// TwinCAT 3 PLC project Caller
// ProgramVersion: 3.1.4023.0
// libraries:
//   Tc2_DataExchange, * (Beckhoff Automation GmbH)
//   Tc2_Standard, * (Beckhoff Automation GmbH)
//   Tc2_System, * (Beckhoff Automation GmbH)
//   Tc2_Utilities, * (Beckhoff Automation GmbH)
//   Tc3_Module, * (Beckhoff Automation GmbH)
// project tree:
//   Code/ F_GetAmsNetId.TcPOU (not stored), I_Executable.TcIO (not stored), I_Logger.TcIO (not stored), ST_AdsReadWriteOptions.TcDUT (not stored), ST_SymbolHandle.TcDUT (not stored), ST_SymbolAddress.TcDUT (not stored), T_AdsWrite.TcPOU, T_GetLastMsgLogger.TcPOU, T_ReleaseHandle.TcPOU, T_GetHandle.TcPOU, T_CallMethod.TcPOU, T_AdsReadWrite.TcPOU, T_InvokeRpcMethod.TcPOU
//   / PlcTask.TcTTO
//   POUs/ FB_InvokeRpcMethod.TcPOU, MAIN.TcPOU
// (motion and I/O tree: see PLC project provider)
// real-time tasks:
//   TASK PlcTask: cycle T#10ms, priority 20, ADS port 350
//   TASK PlcTask1: cycle T#10ms, priority 21, ADS port 351

CONFIGURATION Caller
    RESOURCE PLC ON TwinCAT3
        TASK PlcTask(INTERVAL := T#10ms, PRIORITY := 21);
        PROGRAM MAIN WITH PlcTask : MAIN;
    END_RESOURCE
END_CONFIGURATION

// ---- POUs/MAIN.TcPOU
PROGRAM MAIN
VAR
   xCall : BOOL;
   AddParams : M_ADD_Parameters := (A := 40, B := 2);
   MeaningOfLife : LREAL;
	
	
	askForTheOdds : BOOL;
   c3poAddition : M_ADD_Parameters := (A := 3000, B := 720);
   OddsOfNavigatingAnAsteroidField : LREAL;
	C3PO_Says : STRING(255);

   fbRPC : FB_InvokeRpcMethod;
   invokeRpc : T_InvokeRpcMethod;
   xBusy : BOOL;
   xError : BOOL;
   nErrorID : UDINT;
   methodHandle : ST_SymbolHandle;
   taskState : I_Executable;
   invokeDone, invokeError, invokeBusy : BOOL;
	doneRt, errRt, busyRt : R_TRIG;
   logger : T_GetLastMsgLogger;
   firstScan : BOOL := TRUE;
	
	
END_VAR
VAR CONSTANT
	EMPTY_STRING : STRING := '';
	C3PO_ERR_MSG : STRING(255) := 'Sir, I don$'t know where your ship learned to communicate, but it has the most peculiar dialect.';
END_VAR

fbRPC(
	bCall:=xCall , 
	sNetId :='' , 
	nPort :=851 , 
	sMethodName :='MAIN.fbMath#M_ADD' , 
	nSrcAddrParameter :=ADR(AddParams) , 
	nLenParameter :=SIZEOF(AddParams) , 
	nDestAddrReturnValue :=ADR(MeaningOfLife) , 
	nLenReturnValue :=SIZEOF(MeaningOfLife) , 
	tTimeout :=DEFAULT_ADS_TIMEOUT , 
	eComMode :=E_AdsComMode.eAdsComModeFastCom , 
	bBusy =>xBusy , 
	bError =>xError , 
	nErrorId =>nErrorID );

IF firstScan THEN
	firstScan := FALSE;
	invokeRpc.SetLogger(logger);
	
END_IF

logger.lastLog;
logger.lasLogLevel;
C3PO_Says;

invokeRpc();
methodHandle.SymbolAddress.Ads.netId := F_ScanAmsNetIds('0.0.0.0.0.0.0');
methodHandle.SymbolAddress.Ads.port := 851;
methodHandle.SymbolAddress.SymbolName := 'MAIN.fbMath#M_ADD';
methodHandle.SymbolAddress.WriteRef := F_BIGTYPE(pData := ADR(c3poAddition), cbLen := SIZEOF(c3poAddition));
methodHandle.SymbolAddress.ReadRef := F_LREAL(OddsOfNavigatingAnAsteroidField);

IF askForTheOdds THEN
   askForTheOdds := FALSE;
   taskState := 0;

   invokeRpc.TryInvokeMethodCall(
      symbolHandle := methodHandle,
      adsTimeout := DEFAULT_ADS_TIMEOUT,
      status => taskState
   );

END_IF

invokeBusy := taskState <> 0 AND_THEN taskState.Busy;
invokeDone := taskState <> 0 AND_THEN taskState.Done;
invokeError := taskState <> 0 AND_THEN taskState.Error;
busyRt( CLK := invokeBusy );
doneRt( CLK := invokeDone );
errRt( CLK := invokeError);

IF busyRt.Q THEN
	C3PO_Says := EMPTY_STRING;
END_IF

IF doneRt.Q  THEN
	C3PO_Says := CONCAT(
							'Sir, the possibility of successfully navigating an asteroid field is approximately ', 
							CONCAT( TO_STRING(TO_INT(OddsOfNavigatingAnAsteroidField)), ' to 1.')
						);
END_IF

IF errRt.Q  THEN
	C3PO_Says := C3PO_ERR_MSG;
END_IF

END_PROGRAM

// ---- POUs/FB_InvokeRpcMethod.TcPOU
{attribute 'hide_all_locals'}
FUNCTION_BLOCK FB_InvokeRpcMethod
VAR_INPUT
	bCall					: BOOL;
	sNetId					: T_AmsNetId;
	nPort					: T_AmsPort := 851;
	sMethodName				: STRING(255); //Example:MAIN.fbMath#M_ADD
	nSrcAddrParameter		: PVOID;
	nLenParameter			: UDINT;
	                          
	nDestAddrReturnValue	: PVOID;
	nLenReturnValue			: UDINT;
	                          
	tTimeout				: TIME := DEFAULT_ADS_TIMEOUT;
	eComMode				: E_AdsComMode := eAdsComModeSecureCom;
END_VAR                       
VAR_OUTPUT                    
	bBusy					: BOOL;
	bError					: BOOL;
	nErrorId				: UDINT;
END_VAR                       
VAR                           
	_sNetId					: T_AmsNetId;
 	_sMethodName			: STRING(255);	
	_nPort					: T_AmsPort;
	fbGetHandle				: ADSRDWRT;
	fbCallMethod			: ADSRDWRT;
	fbReleaseHandle			: ADSWRITE;
	trigCall				: R_TRIG;
	eStep,eNextStep			: (IDLE,GET_HANDLE,CALL_METHOD,RELEASE_HANDLE) :=IDLE ;
	nMethodHandle 			: DWORD := 0;
END_VAR

trigCall(CLK:=bCall);
CASE eStep OF
	IDLE:
		IF trigCall.Q THEN
			bBusy 				:= TRUE;
			nErrorId 			:= 0;
			bError 				:= FALSE;
			fbGetHandle			(WRTRD := FALSE);
			fbCallMethod		(WRTRD := FALSE);
			fbReleaseHandle		(WRITE := FALSE);
			IF nMethodHandle <> 0 THEN
				IF 	_sMethodName =  sMethodName AND
					_sNetId 	 = 	sNetId 		AND
					_nPort 		 = 	nPort
				THEN
					eStep			:= CALL_METHOD;
				ELSE        	
					eStep			:= RELEASE_HANDLE;
					eNextStep		:= GET_HANDLE;
				END_IF
			ELSE
				eStep	:=GET_HANDLE;
			END_IF
		ELSE
			bBusy := FALSE;
		END_IF
		
	GET_HANDLE:
		fbGetHandle(NETID 		:= sNetId,
					PORT 		:= nPort,
					IDXGRP 		:= ADSIGRP_SYM_HNDBYNAME,
					IDXOFFS 	:= 0,
					SRCADDR 	:= ADR(sMethodName),
					WRITELEN 	:= TO_UDINT(LEN(sMethodName)),
					DESTADDR 	:= ADR(nMethodHandle),
					READLEN 	:= SIZEOF(nMethodHandle),
					WRTRD 		:= TRUE,
					TMOUT 		:= tTimeout,
					ERR 		=> bError,
					ERRID 		=> nErrorId);

		IF NOT fbGetHandle.BUSY THEN
			IF NOT bError THEN
				_sMethodName 	:= sMethodName;
				_sNetId 		:= sNetId;
				_nPort 			:= nPort;
				eStep			:= CALL_METHOD;
			ELSE
				eStep			:= IDLE;
			END_IF
			fbGetHandle(WRTRD := FALSE);
		END_IF
		
	CALL_METHOD:
		fbCallMethod( NETID		:= sNetId , 
					  PORT		:= nPort , 
					  IDXGRP	:= ADSIGRP_SYM_VALBYHND , 
					  IDXOFFS	:= nMethodHandle , 
					  WRITELEN	:= nLenParameter , 
					  READLEN	:= nLenReturnValue , 
					  SRCADDR	:= nSrcAddrParameter , 
					  DESTADDR	:= nDestAddrReturnValue , 
					  WRTRD		:= TRUE , 
					  TMOUT		:= tTimeout , 
					  ERR		=> bError , 
					  ERRID		=> nErrorId );

		IF NOT fbCallMethod.Busy THEN
			IF NOT bError THEN
				IF (eComMode = eAdsComModeSecureCom) THEN
					eStep		:= RELEASE_HANDLE;
					eNextStep	:= IDLE;
				ELSE
					eStep		:= IDLE;
				END_IF
			ELSE
				eStep			:= RELEASE_HANDLE;
				eNextStep		:= IDLE;				
			END_IF
			fbCallMethod(WRTRD := FALSE);
		END_IF							 
							 
							 
	RELEASE_HANDLE:
		fbReleaseHandle(NETID 		:= sNetId,
						PORT 		:= nPort,
						IDXGRP 		:= ADSIGRP_SYM_RELEASEHND,
						IDXOFFS 	:= 0,
            SRCADDR := ADR(nMethodHandle),
            LEN := SIZEOF(nMethodHandle),
						LEN 		:= 0,
						WRITE 		:= TRUE,
						TMOUT 		:= tTimeout,
						ERR 		=> bError,
						ERRID 		=> nErrorId);

		IF NOT fbReleaseHandle.Busy THEN
			nMethodHandle 	:= 0;
			fbReleaseHandle	(Write := FALSE);
			eStep 			:= eNextStep;
		END_IF
	
END_CASE

END_FUNCTION_BLOCK

// ---- Code/T_InvokeRpcMethod.TcPOU
FUNCTION_BLOCK T_InvokeRpcMethod
VAR_INPUT
   bCall : BOOL;
   sNetId : T_AmsNetId;
   nPort : T_AmsPort := 851;
   sMethodName : STRING(255); //Example:MAIN.fbMath#M_ADD
   nSrcAddrParameter : PVOID;
   nLenParameter : UDINT;

   nDestAddrReturnValue : PVOID;
   nLenReturnValue : UDINT;

   tTimeout : TIME := DEFAULT_ADS_TIMEOUT;
   eComMode : E_AdsComMode := eAdsComModeSecureCom;
END_VAR
VAR_OUTPUT
   bBusy : BOOL;
   bError : BOOL;
   nErrorId : UDINT;
END_VAR
VAR
   getHandle : T_GetHandle;
   callMethod : T_CallMethod;
   releaseHandle : T_ReleaseHandle;
   symbolHandle : ST_SymbolHandle;

   _sNetId : T_AmsNetId;
   _sMethodName : STRING(255);
   _nPort : T_AmsPort;
   //	fbGetHandle				: ADSRDWRT;
   //	fbCallMethod			: ADSRDWRT;
   //	fbReleaseHandle			: ADSWRITE;
   trigCall : R_TRIG;
   eStep, prevStep : (
      IDLE,
      GET_HANDLE,
      CALL_METHOD,
      RELEASE_HANDLE
   ) := IDLE;
  status : I_Executable;
END_VAR

trigCall(CLK := bCall);

CASE eStep OF
   IDLE:
	
		prevStep := eStep;
      IF trigCall.Q THEN
         bBusy := TRUE;
         nErrorId := 0;
         bError := FALSE;
			
			symbolHandle.SymbolAddress.SymbolName := sMethodName;
			symbolHandle.Handle := 0;
			symbolHandle.SymbolAddress.Ads.netId := F_ScanAmsNetIds(sNetId);
			symbolHandle.SymbolAddress.Ads.port := nPort;
			
			symbolHandle.SymbolAddress.WriteRef.cbLen := nLenParameter;
			symbolHandle.SymbolAddress.WriteRef.pData := nSrcAddrParameter;
			
			symbolHandle.SymbolAddress.ReadRef.cbLen := nLenReturnValue;
			symbolHandle.SymbolAddress.ReadRef.pData := nDestAddrReturnValue;
			eStep := GET_HANDLE;
         
      ELSE
         bBusy := FALSE;
      END_IF

   GET_HANDLE:
      IF prevStep <> eStep THEN
			getHandle.TryGetHandle(symbolHandle, DEFAULT_ADS_TIMEOUT);
			prevStep := eStep;
			
		ELSE
			IF getHandle.Done THEN
				eStep := CALL_METHOD;
			END_IF
			
		END_IF

   CALL_METHOD:
	
      IF prevStep <> eStep THEN
			callMethod.TryMethodCall(symbolHandle, DEFAULT_ADS_TIMEOUT);
			prevStep := eStep;
			
		ELSE
			IF callMethod.Done THEN
				eStep := RELEASE_HANDLE;
			END_IF
			
		END_IF
      

   RELEASE_HANDLE:
      
		IF prevStep <> eStep THEN
			releaseHandle.TryReleaseHandle(symbolHandle, DEFAULT_ADS_TIMEOUT);
			prevStep := eStep;
			
		ELSE
			IF releaseHandle.Done THEN
				eStep := IDLE;
			END_IF
			
		END_IF

END_CASE

getHandle();
callMethod();
releaseHandle();

END_FUNCTION_BLOCK

// ---- Code/T_GetHandle.TcPOU
FUNCTION_BLOCK T_GetHandle IMPLEMENTS I_Executable
VAR
   logger : I_Logger;
   _symbolHandle : REFERENCE TO ST_SymbolHandle; // just for debug
	readWrite : T_AdsReadWrite;

END_VAR
VAR CONSTANT
   NO_ERR : UDINT := 0;
   LOG_DEBUG : DWORD := 0;
   LOG_INFO : DWORD := ADSLOG_MSGTYPE_HINT;
   LOG_WARNING : DWORD := ADSLOG_MSGTYPE_WARN;
   LOG_ERROR : DWORD := ADSLOG_MSGTYPE_ERROR;
END_VAR

readWrite();

PROPERTY Busy : BOOL
GET
Busy := readWrite.Busy;
END_GET
END_PROPERTY

PROPERTY Done : BOOL
GET
Done := readWrite.Done;
END_GET
END_PROPERTY

PROPERTY Error : BOOL
GET
Error := readWrite.Error;
END_GET
END_PROPERTY

METHOD PRIVATE ToLog
VAR_INPUT
	Msg : STRING(255);
	LogLevel : DWORD; // generic level, can be mapped to logging framework
END_VAR
IF logger = 0 THEN
	RETURN;
	
END_IF

logger.ToLog(Msg, LogLevel);
END_METHOD

METHOD TryGetHandle : BOOL
VAR_IN_OUT
	symbolHandle : ST_SymbolHandle; // This handle object will be used in the next step.
END_VAR
VAR_INPUT
	adsTimeout : TIME := DEFAULT_ADS_TIMEOUT; // DEFAULT_ADS_TIMEOUT is T#5s;
END_VAR
VAR_OUTPUT
	status : I_Executable;
END_VAR
VAR
	readWriteOpts : ST_AdsReadWriteOptions;
END_VAR
VAR CONSTANT
	NO_HANDLE : DWORD := 0;
END_VAR
IF Busy THEN
	ToLog('Cannot TryGetHandle as Busy', LOG_WARNING);
	RETURN;
	
END_IF

_symbolHandle REF= symbolHandle;

readWriteOpts.AdsAddress := symbolHandle.SymbolAddress.Ads;
readWriteOpts.IndexGroup := ADSIGRP_SYM_HNDBYNAME;
readWriteOpts.IndexOffset := 0;
readWriteOpts.WriteParams := F_STRING(symbolHandle.SymbolAddress.SymbolName);
readWriteOpts.ReadParams := F_DWORD(symbolHandle.Handle);
readWriteOpts.Timeout := adsTimeout;

TryGetHandle := readWrite.TryRequest( readWriteOpts, status => status );
END_METHOD

END_FUNCTION_BLOCK

// ---- Code/T_AdsReadWrite.TcPOU
FUNCTION_BLOCK T_AdsReadWrite IMPLEMENTS I_Executable
VAR
   logger : I_Logger;
	_readWriteOpts : ST_AdsReadWriteOptions;
	
   readWrite : ADSRDWRT;

   state, prevState : (
      IDLE,
      REQUEST,
      WAIT_FOR_RESPONSE,
      DONE_STATE,
      ERROR_STATE
   );

   lastErrorId : UDINT;

END_VAR
VAR CONSTANT
   NO_ERR : UDINT := 0;
   LOG_DEBUG : DWORD := 0;
   LOG_INFO : DWORD := ADSLOG_MSGTYPE_HINT;
   LOG_WARNING : DWORD := ADSLOG_MSGTYPE_WARN;
   LOG_ERROR : DWORD := ADSLOG_MSGTYPE_ERROR;
END_VAR

CASE state OF

   IDlE:
      IsEntryActionAndLog();

   REQUEST:
      IsEntryActionAndLog();
		
      lastErrorId := NO_ERR;
      readWrite.WRTRD := TRUE;
      state := WAIT_FOR_RESPONSE;

   WAIT_FOR_RESPONSE:
      IsEntryActionAndLog();

      IF readWrite.ERR THEN
         state := ERROR_STATE;

      ELSIF NOT readWrite.BUSY THEN
         state := DONE_STATE;

      END_IF

   DONE_STATE:
      IsEntryActionAndLog();

   ERROR_STATE:
      IF IsEntryActionAndLog() THEN
         lastErrorId := readWrite.ERRID;
			
      END_IF

END_CASE

readWrite.WRTRD R= NOT Busy;
readWrite();

PROPERTY Busy : BOOL
GET
Busy := 
	NOT Done 
	AND NOT Error 
	AND state <> IDLE;
END_GET
END_PROPERTY

PROPERTY Done : BOOL
GET
Done := state = DONE_STATE;
END_GET
END_PROPERTY

PROPERTY Error : BOOL
GET
Error := state = ERROR_STATE;
END_GET
END_PROPERTY

METHOD PRIVATE IsEntryActionAndLog : BOOL
IsEntryActionAndLog := prevState <> state;

// useful to debug state transitions. to avoid "chatter" LogFramework should have runtime log level switches 
// i.e. https://github.com/Intecre/twincat-utils/tree/master/IntecreUtilities/IntecreUtilities/IntecreUtilities/Utilities/Logger
// see also https://github.com/Intecre/twincat-utils/blob/master/IntecreUtilities/IntecreUtilities/IntecreUtilities/Utilities/T_NamedBase.TcPOU
ToLog(
	Msg := CONCAT(CONCAT(TO_STRING(prevState), ' transition to state '), TO_STRING(state)), 
	LogLevel:= LOG_DEBUG
);

prevState := state;
END_METHOD

METHOD PUBLIC SetLogger
VAR_INPUT
	logger : I_Logger;
END_VAR
THIS^.logger := logger;
END_METHOD

METHOD PRIVATE ToLog
VAR_INPUT
	Msg : STRING(255);
	LogLevel : DWORD; // generic level, can be mapped to logging framework
END_VAR
IF logger = 0 THEN
	RETURN;
	
END_IF

logger.ToLog(Msg, LogLevel);
END_METHOD

METHOD TryRequest : BOOL
VAR_INPUT
	readWriteOptions : ST_AdsReadWriteOptions;
END_VAR
VAR_OUTPUT
	status : I_Executable;
END_VAR
VAR CONSTANT
	NO_HANDLE : DWORD := 0;
END_VAR
IF Busy THEN
	ToLog('Cannot TryRequest as Busy', LOG_WARNING);
	RETURN;
	
END_IF

_readWriteOpts := readWriteOptions;
readWrite(
	NETID := F_GetAmsNetId(_readWriteOpts.AdsAddress.netId),
	PORT := _readWriteOpts.AdsAddress.port,
	IDXGRP := _readWriteOpts.IndexGroup,
	IDXOFFS := _readWriteOpts.IndexOffset,
	WRITELEN := _readWriteOpts.WriteParams.cbLen,
	SRCADDR := _readWriteOpts.WriteParams.pData,
	READLEN := _readWriteOpts.ReadParams.cbLen,
	DESTADDR := _readWriteOpts.ReadParams.pData,
	TMOUT := _readWriteOpts.Timeout
);

state := REQUEST;

TryRequest := TRUE;
status := THIS^;
END_METHOD

END_FUNCTION_BLOCK

// ---- Code/T_CallMethod.TcPOU
FUNCTION_BLOCK T_CallMethod IMPLEMENTS I_Executable
VAR
   logger : I_Logger;
	_symbolHandle : ST_SymbolHandle;
	readWrite : T_AdsReadWrite;
END_VAR
VAR CONSTANT
   LOG_DEBUG : DWORD := 0;
   LOG_INFO : DWORD := ADSLOG_MSGTYPE_HINT;
   LOG_WARNING : DWORD := ADSLOG_MSGTYPE_WARN;
   LOG_ERROR : DWORD := ADSLOG_MSGTYPE_ERROR;
END_VAR

readWrite();

PROPERTY Busy : BOOL
GET
Busy := readWrite.Busy;
END_GET
END_PROPERTY

PROPERTY Done : BOOL
GET
Done := readWrite.Done;
END_GET
END_PROPERTY

PROPERTY Error : BOOL
GET
Error := readWrite.Error;
END_GET
END_PROPERTY

METHOD PRIVATE ToLog
VAR_INPUT
	Msg : STRING(255);
	LogLevel : DWORD; // generic level, can be mapped to logging framework
END_VAR
IF logger = 0 THEN
	RETURN;
	
END_IF

logger.ToLog(Msg, LogLevel);
END_METHOD

METHOD TryMethodCall : BOOL
VAR_INPUT
	symbolHandle : ST_SymbolHandle;
	adsTimeout : TIME := DEFAULT_ADS_TIMEOUT; // DEFAULT_ADS_TIMEOUT is T#5s;
END_VAR
VAR_OUTPUT
	status : I_Executable;
END_VAR
VAR
	readWriteOpts : ST_AdsReadWriteOptions;
END_VAR
VAR CONSTANT
	NO_HANDLE : DWORD := 0;
END_VAR
IF Busy THEN
	ToLog('Cannot TryGetHandle as Busy', LOG_WARNING);
	RETURN;
	
END_IF

_symbolHandle := symbolHandle;

readWriteOpts.AdsAddress := _symbolHandle.SymbolAddress.Ads;
readWriteOpts.IndexGroup := ADSIGRP_SYM_VALBYHND;
readWriteOpts.IndexOffset := _symbolHandle.Handle;
readWriteOpts.WriteParams := _symbolHandle.SymbolAddress.WriteRef;
readWriteOpts.ReadParams := _symbolHandle.SymbolAddress.ReadRef;
readWriteOpts.Timeout := adsTimeout;

TryMethodCall := readWrite.TryRequest( readWriteOpts, status => status );
END_METHOD

END_FUNCTION_BLOCK

// ---- Code/T_ReleaseHandle.TcPOU
FUNCTION_BLOCK T_ReleaseHandle IMPLEMENTS I_Executable
VAR
   logger : I_Logger;
	_symbolHandle : ST_SymbolHandle;
	write : T_AdsWrite;
END_VAR
VAR CONSTANT
   LOG_DEBUG : DWORD := 0;
   LOG_INFO : DWORD := ADSLOG_MSGTYPE_HINT;
   LOG_WARNING : DWORD := ADSLOG_MSGTYPE_WARN;
   LOG_ERROR : DWORD := ADSLOG_MSGTYPE_ERROR;
END_VAR

write();

PROPERTY Busy : BOOL
GET
Busy := write.Busy;
END_GET
END_PROPERTY

PROPERTY Done : BOOL
GET
Done := write.Done;
END_GET
END_PROPERTY

PROPERTY Error : BOOL
GET
Error := write.Error;
END_GET
END_PROPERTY

METHOD PUBLIC SetLogger
VAR_INPUT
	logger : I_Logger;
END_VAR
THIS^.logger := logger;
END_METHOD

METHOD PRIVATE ToLog
VAR_INPUT
	Msg : STRING(255);
	LogLevel : DWORD; // generic level, can be mapped to logging framework
END_VAR
IF logger = 0 THEN
	RETURN;
	
END_IF

logger.ToLog(Msg, LogLevel);
END_METHOD

METHOD TryReleaseHandle : BOOL
VAR_INPUT
	symbolHandle : ST_SymbolHandle;
	adsTimeout : TIME := DEFAULT_ADS_TIMEOUT; // DEFAULT_ADS_TIMEOUT is T#5s;
END_VAR
VAR_OUTPUT
	status : I_Executable;
END_VAR
VAR
	readWriteOpts : ST_AdsReadWriteOptions;
END_VAR
VAR CONSTANT
	EMPTY_TARG : T_Arg;
	NO_HANDLE : DWORD := 0;
END_VAR
IF Busy THEN
	ToLog('Cannot TryReleaseHandle as Busy', LOG_WARNING);
	RETURN;
	
END_IF

_symbolHandle := symbolHandle;

readWriteOpts.AdsAddress := _symbolHandle.SymbolAddress.Ads;
readWriteOpts.IndexGroup := ADSIGRP_SYM_RELEASEHND;
readWriteOpts.IndexOffset := 0;
readWriteOpts.WriteParams := F_DWORD(_symbolHandle.Handle);
readWriteOpts.ReadParams := EMPTY_TARG;
readWriteOpts.Timeout := adsTimeout;

TryReleaseHandle := write.TryRequest( readWriteOpts, status => status );
END_METHOD

END_FUNCTION_BLOCK

// ---- Code/T_AdsWrite.TcPOU
FUNCTION_BLOCK T_AdsWrite IMPLEMENTS I_Executable
VAR
   logger : I_Logger;
	_readWriteOpts : ST_AdsReadWriteOptions;
	
  write : ADSWRITE;

   state, prevState : (
      IDLE,
      REQUEST,
      WAIT_FOR_RESPONSE,
      DONE_STATE,
      ERROR_STATE
   );

   lastErrorId : UDINT;

END_VAR
VAR CONSTANT
   NO_ERR : UDINT := 0;
   LOG_DEBUG : DWORD := 0;
   LOG_INFO : DWORD := ADSLOG_MSGTYPE_HINT;
   LOG_WARNING : DWORD := ADSLOG_MSGTYPE_WARN;
   LOG_ERROR : DWORD := ADSLOG_MSGTYPE_ERROR;
END_VAR

CASE state OF

   IDlE:
      IsEntryActionAndLog();

   REQUEST:
      IsEntryActionAndLog();
		
      lastErrorId := NO_ERR;
      write.WRITE := TRUE;
      state := WAIT_FOR_RESPONSE;

   WAIT_FOR_RESPONSE:
      IsEntryActionAndLog();

      IF write.ERR THEN
         state := ERROR_STATE;

      ELSIF NOT write.BUSY THEN
         state := DONE_STATE;

      END_IF

   DONE_STATE:
      IsEntryActionAndLog();

   ERROR_STATE:
      IF IsEntryActionAndLog() THEN
         lastErrorId := write.ERRID;
			
      END_IF

END_CASE

write.WRITE R= NOT Busy;
write();

PROPERTY Busy : BOOL
GET
Busy := 
	NOT Done 
	AND NOT Error 
	AND state <> IDLE;
END_GET
END_PROPERTY

PROPERTY Done : BOOL
GET
Done := state = DONE_STATE;
END_GET
END_PROPERTY

PROPERTY Error : BOOL
GET
Error := state = ERROR_STATE;
END_GET
END_PROPERTY

METHOD PRIVATE IsEntryActionAndLog : BOOL
IsEntryActionAndLog := prevState <> state;

// useful to debug state transitions. to avoid "chatter" LogFramework should have runtime log level switches 
// i.e. https://github.com/Intecre/twincat-utils/tree/master/IntecreUtilities/IntecreUtilities/IntecreUtilities/Utilities/Logger
// see also https://github.com/Intecre/twincat-utils/blob/master/IntecreUtilities/IntecreUtilities/IntecreUtilities/Utilities/T_NamedBase.TcPOU
ToLog(
	Msg := CONCAT(CONCAT(TO_STRING(prevState), ' transition to state '), TO_STRING(state)), 
	LogLevel:= LOG_DEBUG
);

prevState := state;
END_METHOD

METHOD PUBLIC SetLogger
VAR_INPUT
	logger : I_Logger;
END_VAR
THIS^.logger := logger;
END_METHOD

METHOD PRIVATE ToLog
VAR_INPUT
	Msg : STRING(255);
	LogLevel : DWORD; // generic level, can be mapped to logging framework
END_VAR
IF logger = 0 THEN
	RETURN;
	
END_IF

logger.ToLog(Msg, LogLevel);
END_METHOD

METHOD TryRequest : BOOL
VAR_INPUT
	readWriteOptions : ST_AdsReadWriteOptions;
END_VAR
VAR_OUTPUT
	status : I_Executable;
END_VAR
VAR CONSTANT
	NO_HANDLE : DWORD := 0;
END_VAR
IF Busy THEN
	ToLog('Cannot TryRequest as Busy', LOG_WARNING);
	RETURN;
	
END_IF

_readWriteOpts := readWriteOptions;
write(
	NETID := F_GetAmsNetId(_readWriteOpts.AdsAddress.netId),
	PORT := _readWriteOpts.AdsAddress.port,
	IDXGRP := _readWriteOpts.IndexGroup,
	IDXOFFS := _readWriteOpts.IndexOffset,
	LEN := _readWriteOpts.WriteParams.cbLen,
	SRCADDR := _readWriteOpts.WriteParams.pData,
	TMOUT := _readWriteOpts.Timeout
);

state := REQUEST;

TryRequest := TRUE;
status := THIS^;
END_METHOD

END_FUNCTION_BLOCK

// ---- Code/T_GetLastMsgLogger.TcPOU
FUNCTION_BLOCK T_GetLastMsgLogger IMPLEMENTS I_Logger

VAR_OUTPUT
	lastLog : STRING;
	lasLogLevel : DWORD;
END_VAR

METHOD ToLog
VAR_INPUT
	Msg	: STRING(255);
	(* generic level, can be mapped to logging framework*)
	LogLevel	: DWORD;
END_VAR
lastLog := MSg;
lasLogLevel := LogLevel;
END_METHOD

END_FUNCTION_BLOCK
